DATA_BLOCK "DB_Wh_MOL"
{ S7_Optimized_Access := 'FALSE' }
VERSION : 0.1
   STRUCT
      HMI_Word_spare : DWord;
      Tank : Array[1..12] of "UDT_Tank_Full";
   END_STRUCT;


BEGIN

END_DATA_BLOCK

